// ---- VISUs/Visu_Walking_Robot_Reset.TcVIS
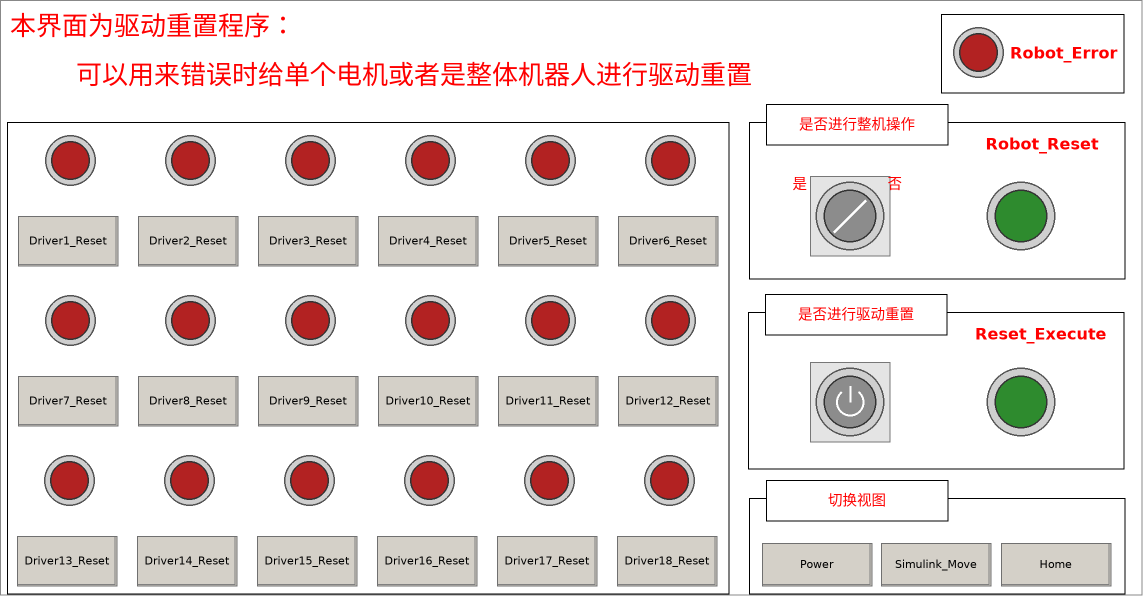
VISUALIZATION Visu_Walking_Robot_Reset  // 1143x596
    Rectangle (7,122 722x472)
    Lamp1 (40,131 61x59), variable: Walking_Robot_Control.Axis_Error[1], style: Lamp-Lamp1-Red
    Lamp1 (160,131 61x59), variable: Walking_Robot_Control.Axis_Error[2], style: Lamp-Lamp1-Red
    Lamp1 (280,131 61x59), variable: Walking_Robot_Control.Axis_Error[3], style: Lamp-Lamp1-Red
    Lamp1 (400,131 61x59), variable: Walking_Robot_Control.Axis_Error[4], style: Lamp-Lamp1-Red
    Lamp1 (520,131 61x59), variable: Walking_Robot_Control.Axis_Error[5], style: Lamp-Lamp1-Red
    Lamp1 (640,131 61x59), variable: Walking_Robot_Control.Axis_Error[6], style: Lamp-Lamp1-Red
    Button (18,216 100x50), "Driver1_Reset"
        tap Walking_Robot_Control.Axis_Reset[1]
    Button (138,216 100x50), "Driver2_Reset"
        tap Walking_Robot_Control.Axis_Reset[2]
    Button (258,216 100x50), "Driver3_Reset"
        tap Walking_Robot_Control.Axis_Reset[3]
    Button (378,216 100x50), "Driver4_Reset"
        tap Walking_Robot_Control.Axis_Reset[4]
    Button (498,216 100x50), "Driver5_Reset"
        tap Walking_Robot_Control.Axis_Reset[5]
    Button (618,216 100x50), "Driver6_Reset"
        tap Walking_Robot_Control.Axis_Reset[6]
    Lamp1 (40,291 61x59), variable: Walking_Robot_Control.Axis_Error[7], style: Lamp-Lamp1-Red
    Lamp1 (160,291 61x59), variable: Walking_Robot_Control.Axis_Error[8], style: Lamp-Lamp1-Red
    Lamp1 (280,291 61x59), variable: Walking_Robot_Control.Axis_Error[9], style: Lamp-Lamp1-Red
    Lamp1 (400,291 61x59), variable: Walking_Robot_Control.Axis_Error[10], style: Lamp-Lamp1-Red
    Lamp1 (520,291 61x59), variable: Walking_Robot_Control.Axis_Error[11], style: Lamp-Lamp1-Red
    Lamp1 (640,291 61x59), variable: Walking_Robot_Control.Axis_Error[12], style: Lamp-Lamp1-Red
    Button (18,376 100x50), "Driver7_Reset"
        tap Walking_Robot_Control.Axis_Reset[7]
    Button (138,376 100x50), "Driver8_Reset"
        tap Walking_Robot_Control.Axis_Reset[8]
    Button (258,376 100x50), "Driver9_Reset"
        tap Walking_Robot_Control.Axis_Reset[9]
    Button (378,376 100x50), "Driver10_Reset"
        tap Walking_Robot_Control.Axis_Reset[10]
    Button (498,376 100x50), "Driver11_Reset"
        tap Walking_Robot_Control.Axis_Reset[11]
    Button (618,376 100x50), "Driver12_Reset"
        tap Walking_Robot_Control.Axis_Reset[12]
    Lamp1 (39,451 61x59), variable: Walking_Robot_Control.Axis_Error[13], style: Lamp-Lamp1-Red
    Lamp1 (159,451 61x59), variable: Walking_Robot_Control.Axis_Error[14], style: Lamp-Lamp1-Red
    Lamp1 (279,451 61x59), variable: Walking_Robot_Control.Axis_Error[15], style: Lamp-Lamp1-Red
    Lamp1 (399,451 61x59), variable: Walking_Robot_Control.Axis_Error[16], style: Lamp-Lamp1-Red
    Lamp1 (519,451 61x59), variable: Walking_Robot_Control.Axis_Error[17], style: Lamp-Lamp1-Red
    Lamp1 (639,451 61x59), variable: Walking_Robot_Control.Axis_Error[18], style: Lamp-Lamp1-Red
    Button (17,536 100x50), "Driver13_Reset"
        tap Walking_Robot_Control.Axis_Reset[13]
    Button (137,536 100x50), "Driver14_Reset"
        tap Walking_Robot_Control.Axis_Reset[14]
    Button (257,536 100x50), "Driver15_Reset"
        tap Walking_Robot_Control.Axis_Reset[15]
    Button (377,536 100x50), "Driver16_Reset"
        tap Walking_Robot_Control.Axis_Reset[16]
    Button (497,536 100x50), "Driver17_Reset"
        tap Walking_Robot_Control.Axis_Reset[17]
    Button (617,536 100x50), "Driver18_Reset"
        tap Walking_Robot_Control.Axis_Reset[18]
    Rectangle (749,122 376x157)
    Label (965,128 154x32), "Robot_Reset"
    Rectangle (766,104 182x41), "是否进行整机操作"
    Rectangle (748,312 376x157)
    Label (964,318 154x32), "Reset_Execute"
    Rectangle (765,294 182x41), "是否进行驱动重置"
    Lamp1 (981,176 80x80), variable: Walking_Robot_Control.Robot_Reset, style: Lamp-Lamp1-Green
    Lamp1 (981,362 80x80), variable: Walking_Robot_Control.Reset_Execute, style: Lamp-Lamp1-Green
    RotarySwitch (810,176 80x80), variable: Walking_Robot_Control.Robot_Reset, behaviour: TOGGLE, style: Switch-RotarySwitch-Gray
    Rectangle (749,498 376x96)
    Rectangle (766,480 182x41), "切换视图"
    Label (865,169 60x30), "否"
    Label (770,169 60x30), "是"
    PowerSwitch (810,362 80x80), variable: Walking_Robot_Control.Reset_Execute, behaviour: TOGGLE, style: Switch-PowerSwitch-Gray
    Label (7,5 365x42), "本界面为驱动重置程序："
    Label (73,54 874x42), "可以用来错误时给单个电机或者是整体机器人进行驱动重置"
    Rectangle (941,14 183x79)
    Lamp1 (948,23 61x59), variable: Walking_Robot_Control.Robot_Error, style: Lamp-Lamp1-Red
    Label (987,37 154x32), "Robot_Error"
    Button (762,543 110x43), "Power"
        OnMouseClick: change screen: Visu_Walking_Robot_Power
    Button (1001,543 110x43), "Home"
        OnMouseClick: change screen: Visu_Walking_Robot_Home
    Button (881,543 110x43), "Simulink_Move"
        OnMouseClick: change screen: Visu_Walking_Robot_SimulinkMove
END_VISUALIZATION

// ---- VISUs/Visu_Walking_Robot_SimulinkMove.TcVIS
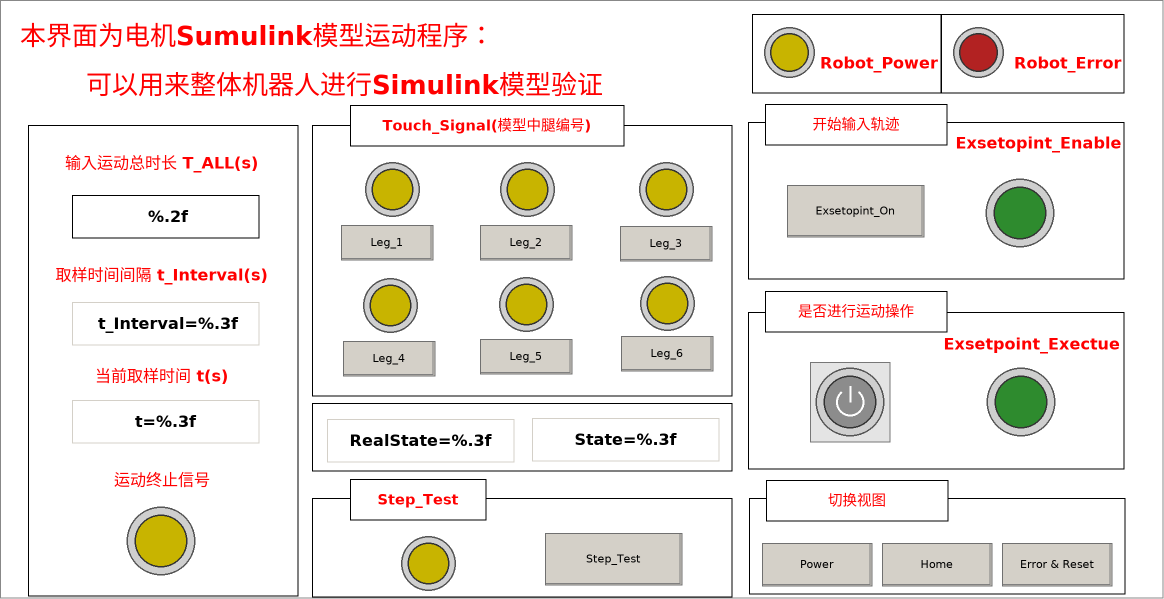
VISUALIZATION Visu_Walking_Robot_SimulinkMove  // 1164x599
    Rectangle (312,498 420x99)
    Rectangle (749,498 376x96)
    Rectangle (766,480 182x41), "切换视图"
    Button (762,543 110x43), "Power"
        OnMouseClick: change screen: Visu_Walking_Robot_Power
    Button (1002,543 110x43), "Error & Reset"
        OnMouseClick: change screen: Visu_Walking_Robot_Reset
    Button (882,543 110x43), "Home"
        OnMouseClick: change screen: Visu_Walking_Robot_Home
    Rectangle (28,125 270x471)
    Rectangle (752,14 189x79)
    Rectangle (748,312 376x157)
    Label (902,328 260x32), "Exsetpoint_Exectue"
    Rectangle (765,291 182x41), "是否进行运动操作"
    Lamp1 (981,362 80x80), variable: Walking_Robot_Movement.ExSetPoint_Execute, style: Lamp-Lamp1-Green
    PowerSwitch (810,362 80x80), variable: Walking_Robot_Movement.ExSetPoint_Execute, behaviour: TOGGLE, style: Switch-PowerSwitch-Gray
    Rectangle (941,14 183x79)
    Lamp1 (948,23 61x59), variable: Walking_Robot_Control.Robot_Error, style: Lamp-Lamp1-Red
    Label (991,47 154x32), "Robot_Error"
    Label (17,15 572x42), "本界面为电机Sumulink模型运动程序："
    Label (83,64 874x42), "可以用来整体机器人进行Simulink模型验证"
    Lamp1 (759,23 61x59), variable: Walking_Robot_Control.Robot_Power, style: Lamp-Lamp1-Yellow
    Label (802,47 154x32), "Robot_Power"
    Rectangle (748,122 376x157)
    Rectangle (765,104 182x41), "开始输入轨迹"
    Lamp1 (980,173 80x80), variable: Walking_Robot_Movement.ExtSetPointEnable, style: Lamp-Lamp1-Green
    Label (935,127 207x32), "Exsetopint_Enable"
    Rectangle (72,195 187x43), "%.2f", text variable: Walking_Robot_Movement.T_All
        OnMouseClick: write Walking_Robot_Movement.T_ALL via Default
    Label (32,147 260x32), "输入运动总时长 T_ALL(s)"
    Textfield (72,400 187x43), "t=%.3f", text variable: Walking_Robot_Movement.t
    Label (32,360 260x32), "当前取样时间 t(s)"
    Button (787,185 137x52), "Exsetopint_On"
        toggle Walking_Robot_Movement.ExtSetPointEnable
    Lamp1 (121,501 80x80), variable: Walking_Robot_Movement.ExtSetPointDisable, style: Lamp-Lamp1-Yellow
    Label (32,464 260x32), "运动终止信号"
    Label (32,259 260x32), "取样时间间隔 t_Interval(s)"
    Textfield (72,302 187x43), "t_Interval=%.3f", text variable: Walking_Robot_Movement.t_Interval
        OnMouseClick: write Walking_Robot_Movement.t_Interval via Default
    Rectangle (312,125 420x271)
    Rectangle (350,105 274x41), "Touch_Signal(模型中腿编号)"
    Lamp1 (361,157 63x65), variable: Walking_Robot_Movement.Touch_Signal[1], style: Lamp-Lamp1-Yellow
    Lamp1 (496,157 63x65), variable: Walking_Robot_Movement.Touch_Signal[2], style: Lamp-Lamp1-Yellow
    Lamp1 (635,157 63x65), variable: Walking_Robot_Movement.Touch_Signal[3], style: Lamp-Lamp1-Yellow
    Lamp1 (359,273 63x65), variable: Walking_Robot_Movement.Touch_Signal[4], style: Lamp-Lamp1-Yellow
    Lamp1 (495,272 63x65), variable: Walking_Robot_Movement.Touch_Signal[5], style: Lamp-Lamp1-Yellow
    Lamp1 (636,271 63x65), variable: Walking_Robot_Movement.Touch_Signal[6], style: Lamp-Lamp1-Yellow
    Rectangle (312,403 420x68)
    Textfield (327,419 187x43), "RealState=%.3f", text variable: Walking_Robot_Movement.realState
    Textfield (532,418 187x43), "State=%.3f", text variable: Walking_Robot_Movement.state
    Button (545,533 137x52), "Step_Test"
        toggle Walking_Robot_Movement.Step_Test
    Lamp1 (397,531 63x65), variable: Walking_Robot_Movement.Step_Test, style: Lamp-Lamp1-Yellow
    Rectangle (350,479 136x41), "Step_Test"
    Button (341,225 92x35), "Leg_1"
        toggle Walking_Robot_Movement.Touch_Signal[1]
    Button (480,225 92x35), "Leg_2"
        toggle Walking_Robot_Movement.Touch_Signal[2]
    Button (620,226 92x35), "Leg_3"
        toggle Walking_Robot_Movement.Touch_Signal[3]
    Button (343,341 92x35), "Leg_4"
        toggle Walking_Robot_Movement.Touch_Signal[4]
    Button (480,339 92x35), "Leg_5"
        toggle Walking_Robot_Movement.Touch_Signal[5]
    Button (621,336 92x35), "Leg_6"
        toggle Walking_Robot_Movement.Touch_Signal[6]
END_VISUALIZATION

// ---- VISUs/Visu_Walking_Robot_Stand.TcVIS
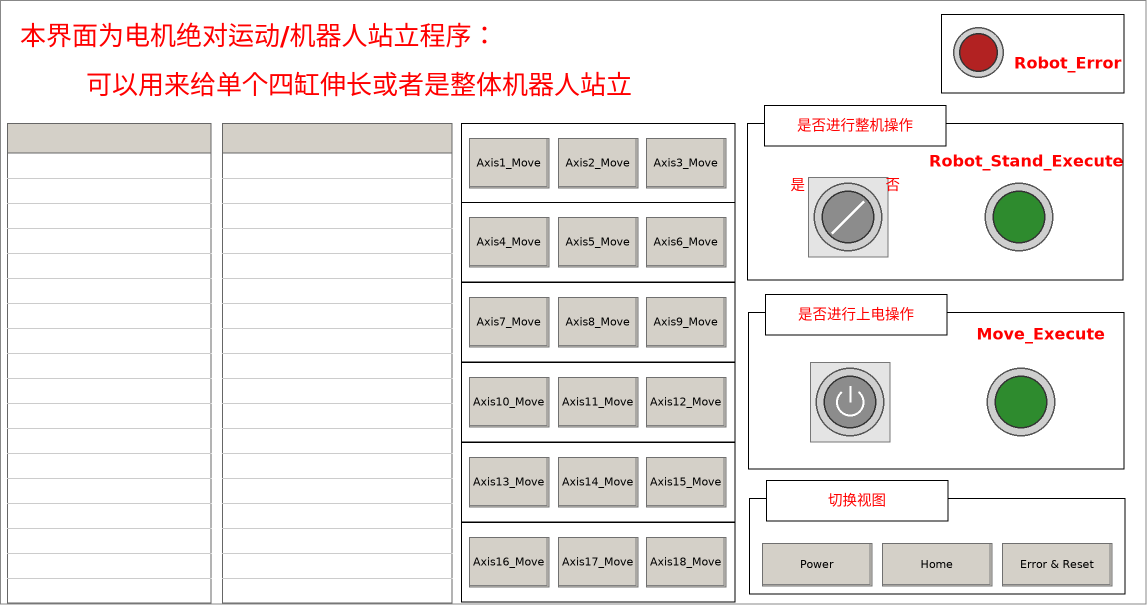
VISUALIZATION Visu_Walking_Robot_Stand  // 1147x605
    Rectangle (941,14 183x79)
    Rectangle (748,312 376x157)
    Label (964,318 154x32), "Move_Execute"
    Rectangle (765,294 182x41), "是否进行上电操作"
    Lamp1 (981,362 80x80), variable: Walking_Robot_Control.Move_Execute, style: Lamp-Lamp1-Green
    PowerSwitch (810,362 80x80), variable: Walking_Robot_Control.Move_Execute, behaviour: TOGGLE, style: Switch-PowerSwitch-Gray
    Lamp1 (948,23 61x59), variable: Walking_Robot_Control.Robot_Error, style: Lamp-Lamp1-Red
    Label (17,15 597x42), "本界面为电机绝对运动/机器人站立程序："
    Label (83,64 719x42), "可以用来给单个四缸伸长或者是整体机器人站立"
    Rectangle (747,123 376x157)
    Rectangle (764,105 182x41), "是否进行整机操作"
    Lamp1 (979,177 80x80), variable: Walking_Robot_Control.Robot_Stand_Execute, style: Lamp-Lamp1-Green
    RotarySwitch (808,177 80x80), variable: Walking_Robot_Control.Robot_Stand_Execute, behaviour: TOGGLE, style: Switch-RotarySwitch-Gray
    Label (863,170 60x30), "否"
    Label (768,170 60x30), "是"
    Label (991,47 154x32), "Robot_Error"
    Table (7,123 204x480), data array: Walking_Robot_Control.Axis_ActPostion
        p3854506369: Walking_Robot_Control.Axis_ActPostion[INDEX]
    Table (222,123 230x480), data array: Walking_Robot_Control.MoveAbsoluteDone
        p3854506369: Walking_Robot_Control.MoveAbsoluteDone[INDEX]
    Rectangle (461,123 274x80)
    Button (469,138 80x50), "Axis1_Move"
        toggle Walking_Robot_Control.Axis_Absolute_Eable[1]
    Button (646,138 80x50), "Axis3_Move"
        toggle Walking_Robot_Control.Axis_Absolute_Eable[3]
    Button (558,138 80x50), "Axis2_Move"
        toggle Walking_Robot_Control.Axis_Absolute_Eable[2]
    Rectangle (461,202 274x80)
    Button (469,217 80x50), "Axis4_Move"
        toggle Walking_Robot_Control.Axis_Absolute_Eable[4]
    Button (646,217 80x50), "Axis6_Move"
        toggle Walking_Robot_Control.Axis_Absolute_Eable[6]
    Button (558,217 80x50), "Axis5_Move"
        toggle Walking_Robot_Control.Axis_Absolute_Eable[5]
    Rectangle (461,282 274x80)
    Button (469,297 80x50), "Axis7_Move"
        toggle Walking_Robot_Control.Axis_Absolute_Eable[7]
    Button (646,297 80x50), "Axis9_Move"
        toggle Walking_Robot_Control.Axis_Absolute_Eable[9]
    Button (558,297 80x50), "Axis8_Move"
        toggle Walking_Robot_Control.Axis_Absolute_Eable[8]
    Rectangle (461,362 274x80)
    Button (469,377 80x50), "Axis10_Move"
        toggle Walking_Robot_Control.Axis_Absolute_Eable[10]
    Button (646,377 80x50), "Axis12_Move"
        toggle Walking_Robot_Control.Axis_Absolute_Eable[12]
    Button (558,377 80x50), "Axis11_Move"
        toggle Walking_Robot_Control.Axis_Absolute_Eable[11]
    Rectangle (461,442 274x80)
    Button (469,457 80x50), "Axis13_Move"
        toggle Walking_Robot_Control.Axis_Absolute_Eable[13]
    Button (646,457 80x50), "Axis15_Move"
        toggle Walking_Robot_Control.Axis_Absolute_Eable[15]
    Button (558,457 80x50), "Axis14_Move"
        toggle Walking_Robot_Control.Axis_Absolute_Eable[14]
    Rectangle (461,522 274x80)
    Button (469,537 80x50), "Axis16_Move"
        toggle Walking_Robot_Control.Axis_Absolute_Eable[16]
    Button (646,537 80x50), "Axis18_Move"
        toggle Walking_Robot_Control.Axis_Absolute_Eable[18]
    Button (558,537 80x50), "Axis17_Move"
        toggle Walking_Robot_Control.Axis_Absolute_Eable[17]
    Label (923,145 207x32), "Robot_Stand_Execute"
    Rectangle (749,498 376x96)
    Rectangle (766,480 182x41), "切换视图"
    Button (762,543 110x43), "Power"
        OnMouseClick: change screen: Visu_Power
    Button (1002,543 110x43), "Error & Reset"
        OnMouseClick: change screen: Visu_Reset
    Button (882,543 110x43), "Home"
        OnMouseClick: change screen: Visu_Home
END_VISUALIZATION

// ---- VISUs/Visu_Walking_Welding_Robot_Control.TcVIS
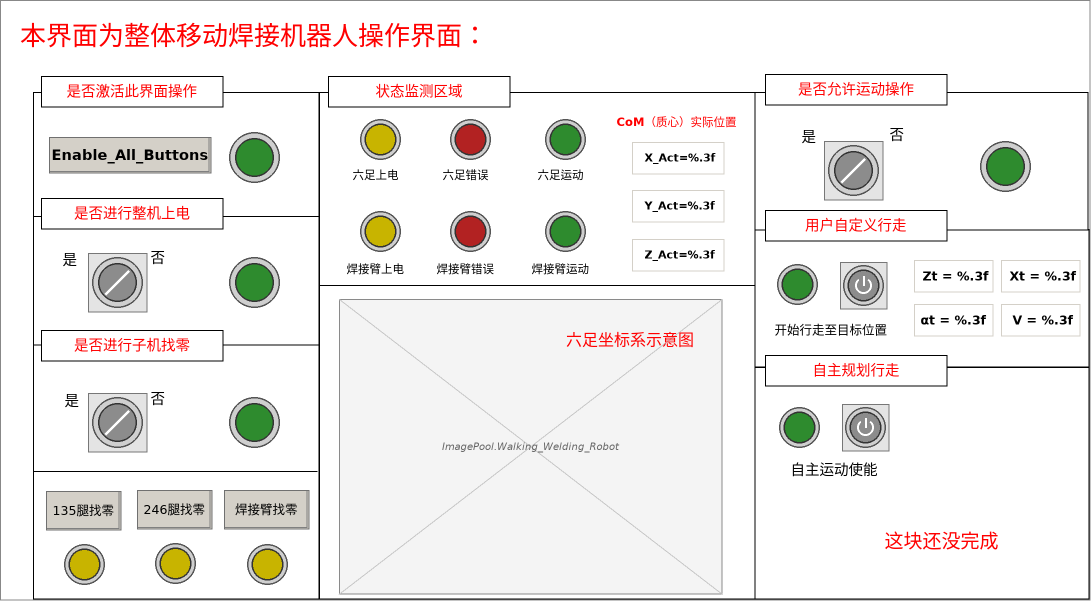
VISUALIZATION Visu_Walking_Welding_Robot_Control  // 1091x601
    Rectangle (754,367 335x232)
    Rectangle (754,229 335x138)
    Rectangle (753,92 335x138)
    Rectangle (33,92 286x125)
    Rectangle (319,92 436x194)
    Rectangle (319,285 436x314)
    Rectangle (33,344 286x255)
    Label (17,15 583x42), "本界面为整体移动焊接机器人操作界面："
    Rectangle (33,216 286x129)
    Lamp1 (225,252 59x61), variable: Walking_Welding_Robot_Control.Walking_Welding_Robot_Power, style: Lamp-Lamp1-Green
    RotarySwitch (88,252 59x61), variable: Walking_Welding_Robot_Control.Walking_Welding_Robot_Power, behaviour: TOGGLE, style: Switch-RotarySwitch-Gray
    Label (138,243 40x30), "否"
    Label (50,245 40x30), "是"
    Rectangle (41,198 182x31), "是否进行整机上电"
    Lamp1 (355,116 51x47), variable: Walking_Robot_Control.Robot_Power, style: Lamp-Lamp1-Yellow
    Lamp1 (445,116 51x47), variable: Walking_Robot_Control.Robot_Error, style: Lamp-Lamp1-Red
    Label (422,159 87x32), "六足错误"
    Label (332,159 87x32), "六足上电"
    Lamp1 (445,208 51x47), variable: Welding_Arm_Control.Welding_Arm_Error, style: Lamp-Lamp1-Red
    Label (422,253 87x32), "焊接臂错误"
    Lamp1 (355,208 51x47), variable: Welding_Arm_Control.Welding_Arm_Power, style: Lamp-Lamp1-Yellow
    Label (332,253 87x32), "焊接臂上电"
    RotarySwitch (88,392 59x61), variable: Walking_Welding_Robot_Control.Walking_Welding_Robot_Home_Execute, behaviour: TOGGLE, style: Switch-RotarySwitch-Gray
    Rectangle (41,330 182x31), "是否进行子机找零"
    Lamp1 (225,392 59x61), variable: Walking_Welding_Robot_Control.Walking_Welding_Robot_Home_Execute, style: Lamp-Lamp1-Green
    Label (138,384 40x30), "否"
    Label (52,386 40x30), "是"
    Rectangle (765,74 182x31), "是否允许运动操作"
    Lamp1 (976,136 59x61), variable: Walking_Welding_Robot_Control.Walking_Welding_Robot_Moving_Execute, style: Lamp-Lamp1-Green
    Button (137,490 75x39), "246腿找零"
        tap Walking_Robot_Control.Leg_Home_Set[2]
    Button (46,491 75x39), "135腿找零"
        tap Walking_Robot_Control.Leg_Home_Set[1]
    Button (224,490 85x39), "焊接臂找零"
        tap Welding_Arm_Control.Welding_Arm_Home_Set
    Lamp1 (59,541 51x47), variable: Walking_Robot_Control.Tripod_Home_Done[1], style: Lamp-Lamp1-Yellow
    Lamp1 (150,540 51x47), variable: Walking_Robot_Control.Tripod_Home_Done[2], style: Lamp-Lamp1-Yellow
    Rectangle (765,210 182x31), "用户自定义行走"
    Textfield (914,260 79x32), "Zt = %.3f", text variable: Walking_Welding_Robot_Control.Robot_Walking_Z
        OnMouseClick: write  via Default
    Textfield (1001,260 79x32), "Xt = %.3f", text variable: Walking_Welding_Robot_Control.Robot_Walking_X
        OnMouseClick: write  via Default
    Textfield (914,304 79x32), "αt = %.3f", text variable: Walking_Welding_Robot_Control.Robot_Walking_alpha
        OnMouseClick: write  via Default
    Textfield (1001,304 79x32), "V = %.3f", text variable: Walking_Welding_Robot_Control.Robot_Walking_Velocity
        OnMouseClick: write  via Default
    Lamp1 (772,261 51x47), variable: Walking_Welding_Robot_Control.User_Moving_Control, style: Lamp-Lamp1-Green
    PowerSwitch (838,262 51x47), variable: Walking_Welding_Robot_Control.User_Moving_Control, behaviour: TOGGLE, style: Switch-PowerSwitch-Gray
    Image (339,299 383x295), image: ImagePool.Walking_Welding_Robot
    Textfield (632,239 92x32), "Z_Act=%.3f", text variable: Walking_Robot_Movement.Act_Slice[3]
    Textfield (632,142 92x32), "X_Act=%.3f", text variable: Walking_Robot_Movement.Act_Slice[4]
    Textfield (632,190 92x32), "Y_Act=%.3f", text variable: Walking_Robot_Movement.Act_Slice[5]
    Lamp1 (540,116 51x47), variable: Walking_Robot_Movement.ExtSetPointEnable, style: Lamp-Lamp1-Green
    Lamp1 (540,208 51x47), variable: Welding_Arm_Movement.ExtSetPointEnable, style: Lamp-Lamp1-Green
    Label (517,159 87x32), "六足运动"
    Label (517,253 87x32), "焊接臂运动"
    Rectangle (765,355 182x31), "自主规划行走"
    PowerSwitch (840,404 51x47), variable: Walking_Welding_Robot_Control.Auto_Moving_Control, behaviour: TOGGLE, style: Switch-PowerSwitch-Gray
    Lamp1 (774,404 51x47), variable: Walking_Welding_Robot_Control.Auto_Moving_Control, style: Lamp-Lamp1-Green
    Label (781,454 106x32), "自主运动使能"
    Button (49,137 162x36), "Enable_All_Buttons"
        toggle Walking_Welding_Robot_Control.Walking_Welding_Robot_Joint_Control
    Lamp1 (225,127 59x61), variable: Walking_Welding_Robot_Control.Walking_Welding_Robot_Joint_Control, style: Lamp-Lamp1-Green
    Label (759,314 144x32), "开始行走至目标位置"
    Line (33,471) (317,471)
    Rectangle (328,76 182x31), "状态监测区域"
    Rectangle (41,76 182x31), "是否激活此界面操作"
    Label (526,325 208x30), "六足坐标系示意图"
    Label (603,107 147x30), "CoM（质心）实际位置"
    Label (877,120 40x30), "否"
    Label (789,122 40x30), "是"
    RotarySwitch (824,140 59x61), variable: Walking_Welding_Robot_Control.Walking_Welding_Robot_Moving_Execute, behaviour: TOGGLE, style: Switch-RotarySwitch-Gray
    Label (851,525 181x32), "这块还没完成"
    Lamp1 (242,541 51x47), variable: Welding_Arm_Control.Welding_Arm_Home_Done, style: Lamp-Lamp1-Yellow
END_VISUALIZATION

// ---- VISUs/Visu_Welcome.TcVIS
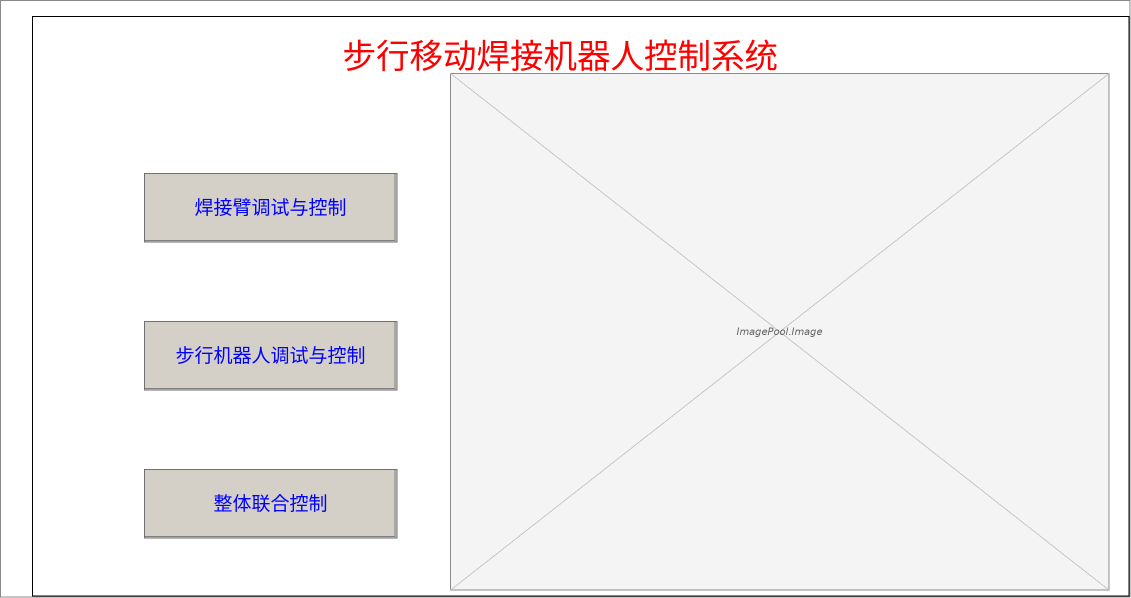
VISUALIZATION Visu_Welcome  // 1131x598
    Rectangle (32,16 1097x580)
    Image (716,328 150x30)
    Label (269,35 583x42), "步行移动焊接机器人控制系统"
    Button (144,469 253x69), "整体联合控制"
        OnMouseClick: change screen: Visu_Walking_Welding_Robot_Control
    Button (144,321 253x69), "步行机器人调试与控制"
        OnMouseClick: change screen: Visu_Walking_Robot_Power
    Button (144,173 253x69), "焊接臂调试与控制"
        OnMouseClick: change screen: Visu_Welding_Arm_Power
    Image (450,73 659x517), image: ImagePool.Image
END_VISUALIZATION

// ---- VISUs/Visu_Welding_Arm_OldVersion.TcVIS
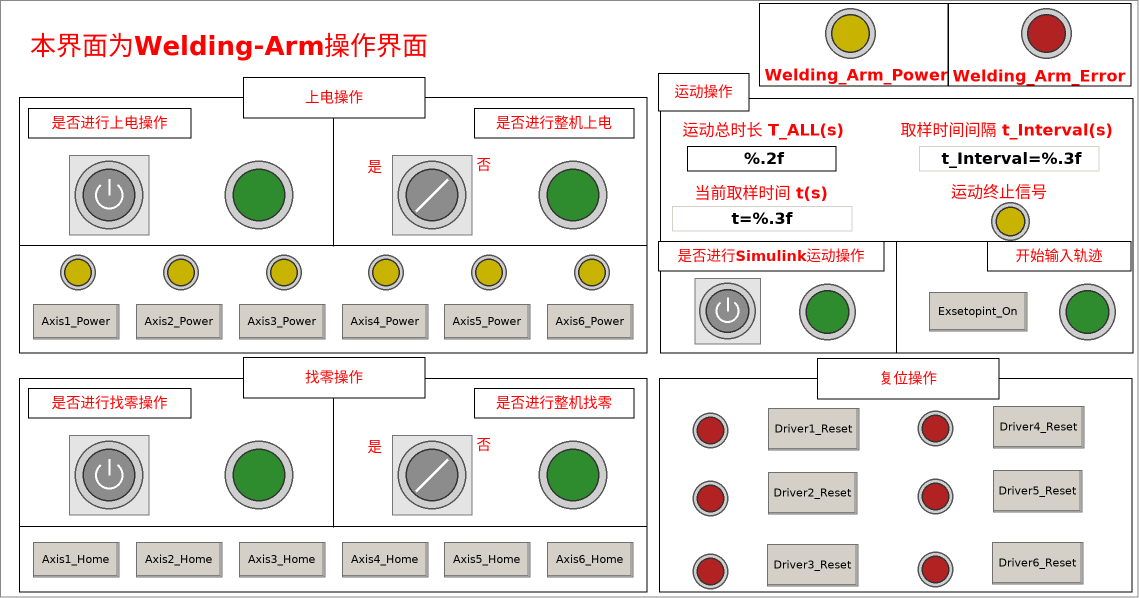
VISUALIZATION Visu_Welding_Arm_OldVersion  // 1139x598
    Rectangle (660,98 473x255)
    Rectangle (659,378 473x214)
    Group (19,97 628x256)
        Rectangle (0,0 628x256)
        Line (1,148) (627,148)
        Line (314,0) (314,149)
    Label (345,152 60x30), "是"
    Label (454,150 60x30), "否"
    Rectangle (474,108 160x30), "是否进行整机上电"
    Lamp1 (219,155 80x80), variable: Welding_Arm_Control.Power_Execute, style: Lamp-Lamp1-Green
    Lamp1 (52,252 52x41), variable: Welding_Arm_Control.Power_Status[1], style: Lamp-Lamp1-Yellow
    Lamp1 (155,252 52x41), variable: Welding_Arm_Control.Power_Status[2], style: Lamp-Lamp1-Yellow
    Lamp1 (258,252 52x41), variable: Welding_Arm_Control.Power_Status[3], style: Lamp-Lamp1-Yellow
    Lamp1 (360,252 52x41), variable: Welding_Arm_Control.Power_Status[4], style: Lamp-Lamp1-Yellow
    Lamp1 (463,252 52x41), variable: Welding_Arm_Control.Power_Status[5], style: Lamp-Lamp1-Yellow
    Lamp1 (566,252 52x41), variable: Welding_Arm_Control.Power_Status[6], style: Lamp-Lamp1-Yellow
    Button (33,304 86x35), "Axis1_Power"
        toggle Welding_Arm_Control.Axis_Power[1]
    Button (136,304 86x35), "Axis2_Power"
        toggle Welding_Arm_Control.Axis_Power[2]
    Button (239,304 86x35), "Axis3_Power"
        toggle Welding_Arm_Control.Axis_Power[3]
    Button (342,304 86x35), "Axis4_Power"
        toggle Welding_Arm_Control.Axis_Power[4]
    Button (444,304 86x35), "Axis5_Power"
        toggle Welding_Arm_Control.Axis_Power[5]
    Button (547,304 86x35), "Axis6_Power"
        toggle Welding_Arm_Control.Axis_Power[6]
    Rectangle (28,108 163x30), "是否进行上电操作"
    PowerSwitch (69,155 80x80), variable: Welding_Arm_Control.Power_Execute, behaviour: TOGGLE, style: Switch-PowerSwitch-Gray
    Lamp1 (533,155 80x80), variable: Welding_Arm_Control.Robot_Power, style: Lamp-Lamp1-Green
    RotarySwitch (392,155 80x80), variable: Welding_Arm_Control.Welding_Arm_Power, behaviour: TOGGLE, style: Switch-RotarySwitch-Gray
    Rectangle (243,77 182x41), "上电操作"
    Group (19,378 628x214)
        Rectangle (0,0 628x214)
        Line (1,148) (627,148)
        Line (314,0) (314,149)
    Label (345,432 60x30), "是"
    Label (454,430 60x30), "否"
    Rectangle (474,388 160x30), "是否进行整机找零"
    Lamp1 (219,435 80x80), variable: Welding_Arm_Control.Power_Execute, style: Lamp-Lamp1-Green
    Button (33,542 86x35), "Axis1_Home"
        toggle Welding_Arm_Control.Axis_Home_Set[1]
    Button (136,542 86x35), "Axis2_Home"
        toggle Welding_Arm_Control.Axis_Home_Set[2]
    Button (239,542 86x35), "Axis3_Home"
        toggle Welding_Arm_Control.Axis_Home_Set[3]
    Button (342,542 86x35), "Axis4_Home"
        toggle Welding_Arm_Control.Axis_Home_Set[4]
    Button (444,542 86x35), "Axis5_Home"
        toggle Welding_Arm_Control.Axis_Home_Set[5]
    Button (547,542 86x35), "Axis6_Home"
        toggle Welding_Arm_Control.Axis_Home_Set[6]
    Rectangle (28,388 163x30), "是否进行找零操作"
    PowerSwitch (69,435 80x80), variable: Welding_Arm_Control.Home_Execute, behaviour: TOGGLE, style: Switch-PowerSwitch-Gray
    Lamp1 (533,435 80x80), variable: Welding_Arm_Control.Robot_Power, style: Lamp-Lamp1-Green
    RotarySwitch (392,435 80x80), variable: Welding_Arm_Control.Welding_Arm_Home_Set, behaviour: TOGGLE, style: Switch-RotarySwitch-Gray
    Rectangle (243,357 182x41), "找零操作"
    Rectangle (759,3 189x83)
    Rectangle (948,3 183x83)
    Lamp1 (1016,4 61x59), variable: Welding_Arm_Control.Robot_Error, style: Lamp-Lamp1-Red
    Label (953,60 172x32), "Welding_Arm_Error"
    Lamp1 (820,4 61x59), variable: Welding_Arm_Control.Robot_Power, style: Lamp-Lamp1-Yellow
    Label (766,59 181x32), "Welding_Arm_Power"
    Lamp1 (690,406 41x49), variable: Welding_Arm_Control.Axis_Error[1], style: Lamp-Lamp1-Red
    Lamp1 (690,474 41x49), variable: Welding_Arm_Control.Axis_Error[2], style: Lamp-Lamp1-Red
    Lamp1 (690,547 41x49), variable: Welding_Arm_Control.Axis_Error[3], style: Lamp-Lamp1-Red
    Button (768,408 91x42), "Driver1_Reset"
        tap Welding_Arm_Control.Axis_Reset[1]
    Button (768,472 89x42), "Driver2_Reset"
        tap Welding_Arm_Control.Axis_Reset[2]
    Button (767,544 91x42), "Driver3_Reset"
        tap Welding_Arm_Control.Axis_Reset[3]
    Lamp1 (915,404 41x49), variable: Welding_Arm_Control.Axis_Error[1], style: Lamp-Lamp1-Red
    Lamp1 (915,472 41x49), variable: Welding_Arm_Control.Axis_Error[2], style: Lamp-Lamp1-Red
    Lamp1 (915,545 41x49), variable: Welding_Arm_Control.Axis_Error[3], style: Lamp-Lamp1-Red
    Button (993,406 91x42), "Driver4_Reset"
        tap Welding_Arm_Control.Axis_Reset[4]
    Button (993,470 89x42), "Driver5_Reset"
        tap Welding_Arm_Control.Axis_Reset[5]
    Button (992,542 91x42), "Driver6_Reset"
        tap Welding_Arm_Control.Axis_Reset[6]
    Rectangle (687,146 149x25), "%.2f", text variable: Welding_Arm_Movement.T_ALL
        OnMouseClick: write Welding_Arm_Movement.T_ALL via Default
    Label (664,118 199x24), "运动总时长 T_ALL(s)"
    Textfield (672,206 180x25), "t=%.3f", text variable: Welding_Arm_Movementl.t
    Label (684,181 155x24), "当前取样时间 t(s)"
    Lamp1 (982,199 57x45), variable: Robot_Movement.ExtSetPointDisable, style: Lamp-Lamp1-Yellow
    Label (909,180 180x24), "运动终止信号"
    Label (877,118 260x24), "取样时间间隔 t_Interval(s)"
    Textfield (919,146 180x25), "t_Interval=%.3f", text variable: Welding_Arm_Movement.t_Interval
        OnMouseClick: write Welding_Arm_Movement.t_Interval via Default
    Rectangle (817,358 182x41), "复位操作"
    Line (659,241) (1131,241)
    Rectangle (658,241 226x30), "是否进行Simulink运动操作"
    Lamp1 (791,279 73x66), variable: Welding_Arm_Movement.ExSetPoint_Execute, style: Lamp-Lamp1-Green
    PowerSwitch (691,278 73x66), variable: Welding_Arm_Movement.ExSetPoint_Execute, behaviour: TOGGLE, style: Switch-PowerSwitch-Gray
    Rectangle (987,241 144x30), "开始输入轨迹"
    Button (929,292 98x39), "Exsetopint_On"
        toggle Welding_Arm_Movement.ExtSetPointEnable
    Lamp1 (1051,279 73x66), variable: Welding_Arm_Movement.ExtSetPointEnable, style: Lamp-Lamp1-Green
    Line (896,242) (896,352)
    Label (27,25 572x42), "本界面为Welding-Arm操作界面"
    Rectangle (658,73 91x38), "运动操作"
END_VISUALIZATION
